PROGRAM POU_AbortMoves
VAR
	fbAxis1Halt:MC_Halt;
	fbAxis2Halt:MC_Halt;
	fbAxis3Halt:MC_Halt;
	fbAxis4Halt:MC_Halt;
	fbAxis5Halt:MC_Halt;
	fbAxis6Halt:MC_Halt;
	
END_VAR

fbAxis1Halt(
	Axis:= , 
	Execute:= , 
	Deceleration:= , 
	Jerk:= , 
	BufferMode:= , 
	Options:= , 
	Done=> , 
	Busy=> , 
	Active=> , 
	CommandAborted=> , 
	Error=> , 
	ErrorID=> );
	
fbAxis2Halt(
	Axis:= , 
	Execute:= , 
	Deceleration:= , 
	Jerk:= , 
	BufferMode:= , 
	Options:= , 
	Done=> , 
	Busy=> , 
	Active=> , 
	CommandAborted=> , 
	Error=> , 
	ErrorID=> );
	
fbAxis3Halt(
	Axis:= , 
	Execute:= , 
	Deceleration:= , 
	Jerk:= , 
	BufferMode:= , 
	Options:= , 
	Done=> , 
	Busy=> , 
	Active=> , 
	CommandAborted=> , 
	Error=> , 
	ErrorID=> );
	
fbAxis4Halt(
	Axis:= , 
	Execute:= , 
	Deceleration:= , 
	Jerk:= , 
	BufferMode:= , 
	Options:= , 
	Done=> , 
	Busy=> , 
	Active=> , 
	CommandAborted=> , 
	Error=> , 
	ErrorID=> );
	
fbAxis5Halt(
	Axis:= , 
	Execute:= , 
	Deceleration:= , 
	Jerk:= , 
	BufferMode:= , 
	Options:= , 
	Done=> , 
	Busy=> , 
	Active=> , 
	CommandAborted=> , 
	Error=> , 
	ErrorID=> );
	
fbAxis6Halt(
	Axis:= , 
	Execute:= , 
	Deceleration:= , 
	Jerk:= , 
	BufferMode:= , 
	Options:= , 
	Done=> , 
	Busy=> , 
	Active=> , 
	CommandAborted=> , 
	Error=> , 
	ErrorID=> );

END_PROGRAM

(* stored: Version 1.1.0.1, ProductVersion 3.1.4022.18
   POU POU_AbortMoves: Id {55d13cdc-4a62-47c8-a724-0abc837a49f9}, SpecialFunc None *)
